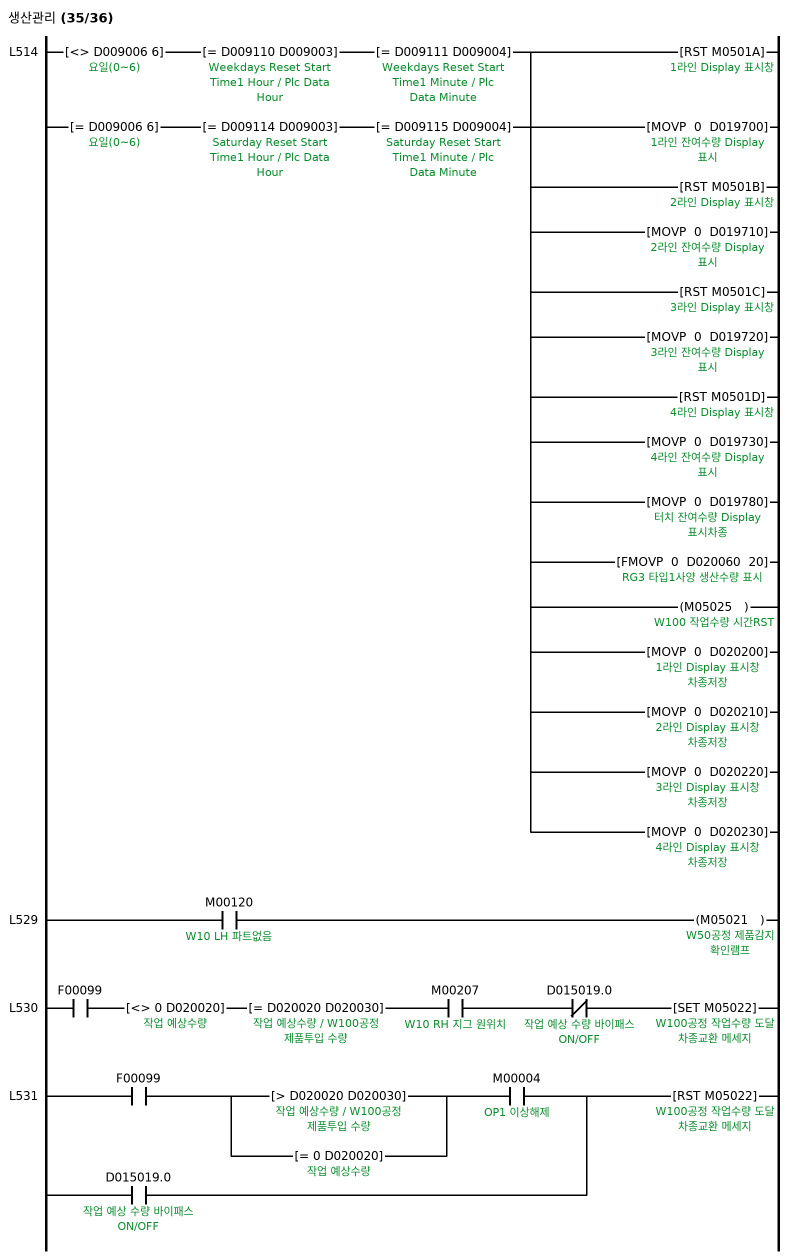
[picture p480: 생산관리 rungs L514-L531]
; L514
LOAD<>    D009006 6	// 요일(0~6)
AND=      D009110 D009003	// Weekdays Reset Start Time1 Hour / Plc Data Hour
AND=      D009111 D009004	// Weekdays Reset Start Time1 Minute / Plc Data Minute
LOAD=     D009006 6	// 요일(0~6)
AND=      D009114 D009003	// Saturday Reset Start Time1 Hour / Plc Data Hour
AND=      D009115 D009004	// Saturday Reset Start Time1 Minute / Plc Data Minute
OR LOAD
RST       M0501A	// 1라인 Display 표시창
MOVP      0 D019700	// 1라인 잔여수량 Display 표시 
RST       M0501B	// 2라인 Display 표시창
MOVP      0 D019710	// 2라인 잔여수량 Display 표시 
RST       M0501C	// 3라인 Display 표시창
MOVP      0 D019720	// 3라인 잔여수량 Display 표시 
RST       M0501D	// 4라인 Display 표시창
MOVP      0 D019730	// 4라인 잔여수량 Display 표시 
MOVP      0 D019780	// 터치 잔여수량 Display 표시차종
FMOVP     0 D020060 20	// RG3 타입1사양 생산수량 표시
OUT       M05025	// W100 작업수량 시간RST
MOVP      0 D020200	// 1라인 Display 표시창 차종저장
MOVP      0 D020210	// 2라인 Display 표시창 차종저장
MOVP      0 D020220	// 3라인 Display 표시창 차종저장
MOVP      0 D020230	// 4라인 Display 표시창 차종저장
; L529
LOAD      M00120	// W10 LH 파트없음
OUT       M05021	// W50공정 제품감지 확인램프
; L530
LOAD      F00099
AND<>     0 D020020	// 작업 예상수량
AND=      D020020 D020030	// 작업 예상수량 / W100공정 제품투입 수량
AND       M00207	// W10 RH 지그 원위치
AND NOT   D015019.0	// 작업 예상 수량 바이패스 ON/OFF
SET       M05022	// W100공정 작업수량 도달 차종교환 메세지
; L531
LOAD      F00099
LOAD>     D020020 D020030	// 작업 예상수량 / W100공정 제품투입 수량
OR=       0 D020020	// 작업 예상수량
AND LOAD
AND       M00004	// OP1 이상해제
OR        D015019.0	// 작업 예상 수량 바이패스 ON/OFF
RST       M05022	// W100공정 작업수량 도달 차종교환 메세지

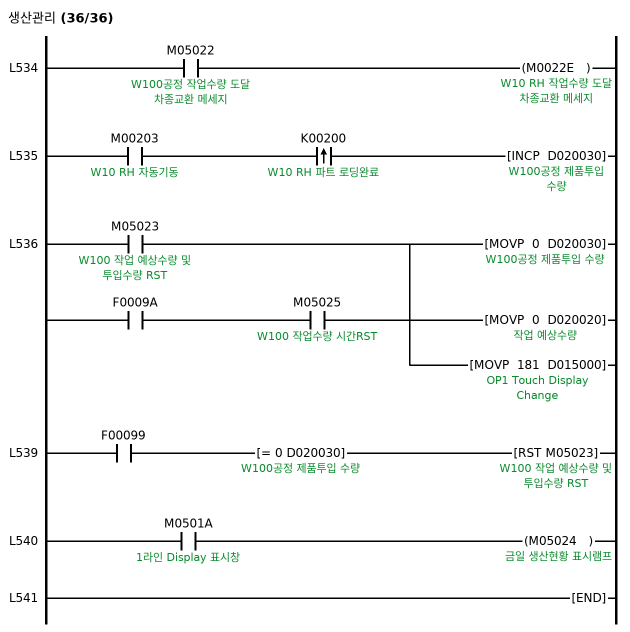
; L534
LOAD      M05022	// W100공정 작업수량 도달 차종교환 메세지
OUT       M0022E	// W10 RH 작업수량 도달 차종교환 메세지
; L535
LOAD      M00203	// W10 RH 자동기동
ANDP      K00200	// W10 RH 파트 로딩완료
INCP      D020030	// W100공정 제품투입 수량
; L536
LOAD      M05023	// W100 작업 예상수량 및 투입수량 RST
LOAD      F0009A
AND       M05025	// W100 작업수량 시간RST
OR LOAD
MOVP      0 D020030	// W100공정 제품투입 수량
MOVP      0 D020020	// 작업 예상수량
MOVP      181 D015000	// OP1 Touch Display Change
; L539
LOAD      F00099
AND=      0 D020030	// W100공정 제품투입 수량
RST       M05023	// W100 작업 예상수량 및 투입수량 RST
; L540
LOAD      M0501A	// 1라인 Display 표시창
OUT       M05024	// 금일 생산현황 표시램프
; L541
END

PROGRAM 생산현황판 (task: 스캔 프로그램)

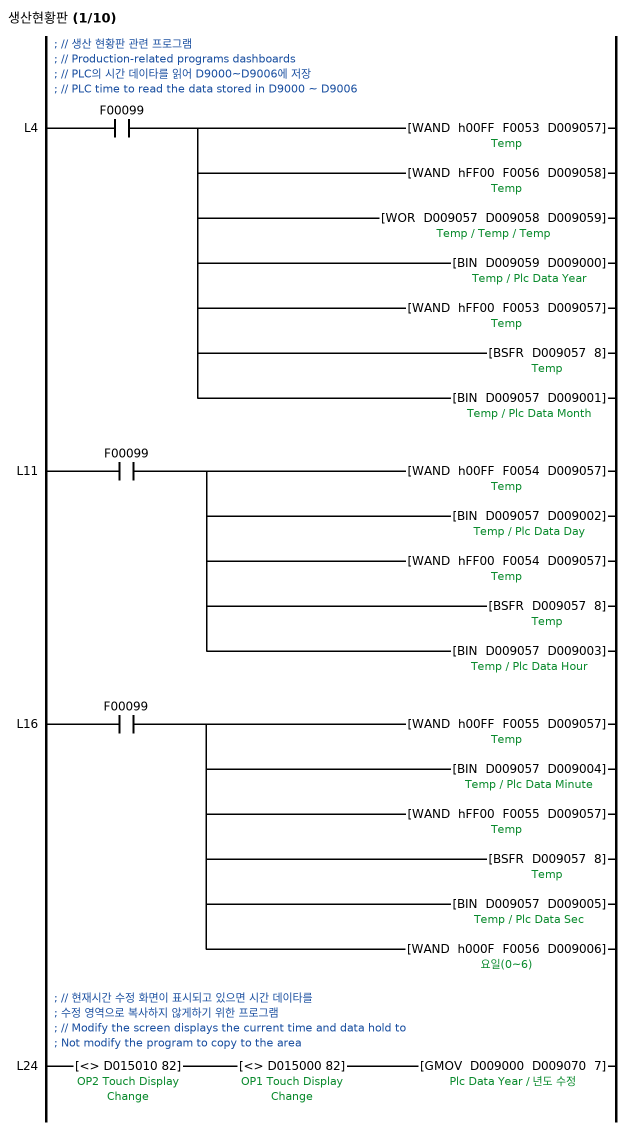
// // 생산 현황판 관련 프로그램
// // Production-related programs dashboards
//   // PLC의 시간 데이타를 읽어 D9000~D9006에 저장
//   // PLC time to read the data stored in D9000 ~ D9006
; L4
LOAD      F00099
WAND      h00FF F0053 D009057	// Temp
WAND      hFF00 F0056 D009058	// Temp
WOR       D009057 D009058 D009059	// Temp / Temp / Temp
BIN       D009059 D009000	// Temp / Plc Data Year
WAND      hFF00 F0053 D009057	// Temp
BSFR      D009057 8	// Temp
BIN       D009057 D009001	// Temp / Plc Data Month
; L11
LOAD      F00099
WAND      h00FF F0054 D009057	// Temp
BIN       D009057 D009002	// Temp / Plc Data Day
WAND      hFF00 F0054 D009057	// Temp
BSFR      D009057 8	// Temp
BIN       D009057 D009003	// Temp / Plc Data Hour
; L16
LOAD      F00099
WAND      h00FF F0055 D009057	// Temp
BIN       D009057 D009004	// Temp / Plc Data Minute
WAND      hFF00 F0055 D009057	// Temp
BSFR      D009057 8	// Temp
BIN       D009057 D009005	// Temp / Plc Data Sec
WAND      h000F F0056 D009006	// 요일(0~6)
//   // 현재시간 수정 화면이 표시되고 있으면 시간 데이타를
//      수정 영역으로 복사하지 않게하기 위한 프로그램
//   // Modify the screen displays the current time and data hold to
//       Not modify the program to copy to the area
; L24
LOAD<>    D015010 82	// OP2 Touch Display Change
AND<>     D015000 82	// OP1 Touch Display Change
GMOV      D009000 D009070 7	// Plc Data Year / 년도 수정

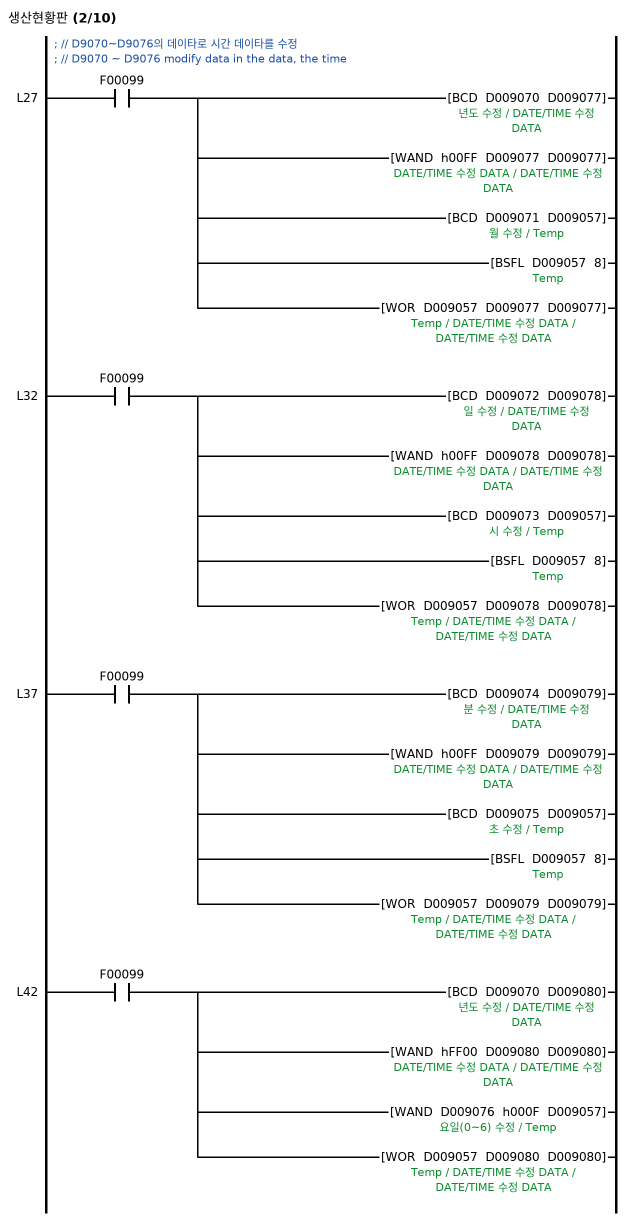
//   // D9070~D9076의 데이타로 시간 데이타를 수정
//   // D9070 ~ D9076 modify data in the data, the time
; L27
LOAD      F00099
BCD       D009070 D009077	// 년도 수정 / DATE/TIME 수정 DATA
WAND      h00FF D009077 D009077	// DATE/TIME 수정 DATA / DATE/TIME 수정 DATA
BCD       D009071 D009057	// 월 수정 / Temp
BSFL      D009057 8	// Temp
WOR       D009057 D009077 D009077	// Temp / DATE/TIME 수정 DATA / DATE/TIME 수정 DATA
; L32
LOAD      F00099
BCD       D009072 D009078	// 일 수정 / DATE/TIME 수정 DATA
WAND      h00FF D009078 D009078	// DATE/TIME 수정 DATA / DATE/TIME 수정 DATA
BCD       D009073 D009057	// 시 수정 / Temp
BSFL      D009057 8	// Temp
WOR       D009057 D009078 D009078	// Temp / DATE/TIME 수정 DATA / DATE/TIME 수정 DATA
; L37
LOAD      F00099
BCD       D009074 D009079	// 분 수정 / DATE/TIME 수정 DATA
WAND      h00FF D009079 D009079	// DATE/TIME 수정 DATA / DATE/TIME 수정 DATA
BCD       D009075 D009057	// 초 수정 / Temp
BSFL      D009057 8	// Temp
WOR       D009057 D009079 D009079	// Temp / DATE/TIME 수정 DATA / DATE/TIME 수정 DATA
; L42
LOAD      F00099
BCD       D009070 D009080	// 년도 수정 / DATE/TIME 수정 DATA
WAND      hFF00 D009080 D009080	// DATE/TIME 수정 DATA / DATE/TIME 수정 DATA
WAND      D009076 h000F D009057	// 요일(0~6) 수정 / Temp
WOR       D009057 D009080 D009080	// Temp / DATE/TIME 수정 DATA / DATE/TIME 수정 DATA

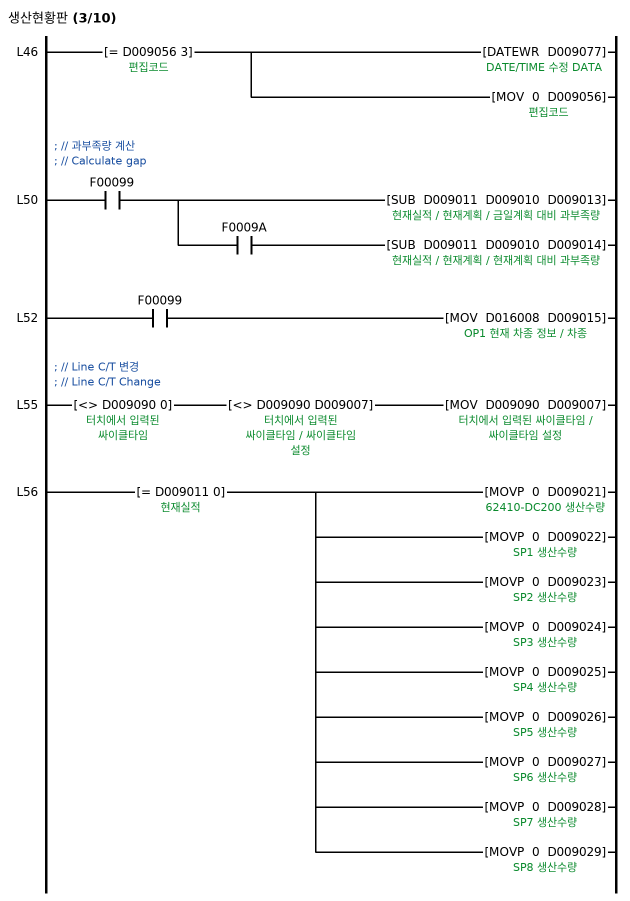
; L46
LOAD=     D009056 3	// 편집코드
DATEWR    D009077	// DATE/TIME 수정 DATA
MOV       0 D009056	// 편집코드
//   // 과부족량 계산
//   // Calculate gap
; L50
LOAD      F00099
SUB       D009011 D009010 D009013	// 현재실적 / 현재계획 / 금일계획 대비 과부족량
AND       F0009A
SUB       D009011 D009010 D009014	// 현재실적 / 현재계획 / 현재계획 대비 과부족량
; L52
LOAD      F00099
MOV       D016008 D009015	// OP1 현재 차종 정보 / 차종
//   // Line C/T 변경
//   // Line C/T Change
; L55
LOAD<>    D009090 0	// 터치에서 입력된 싸이클타임
AND<>     D009090 D009007	// 터치에서 입력된 싸이클타임 / 싸이클타임 설정
MOV       D009090 D009007	// 터치에서 입력된 싸이클타임 / 싸이클타임 설정
; L56
LOAD=     D009011 0	// 현재실적
MOVP      0 D009021	// 62410-DC200 생산수량
MOVP      0 D009022	// SP1 생산수량
MOVP      0 D009023	// SP2 생산수량
MOVP      0 D009024	// SP3 생산수량
MOVP      0 D009025	// SP4 생산수량
MOVP      0 D009026	// SP5 생산수량
MOVP      0 D009027	// SP6 생산수량
MOVP      0 D009028	// SP7 생산수량
MOVP      0 D009029	// SP8 생산수량

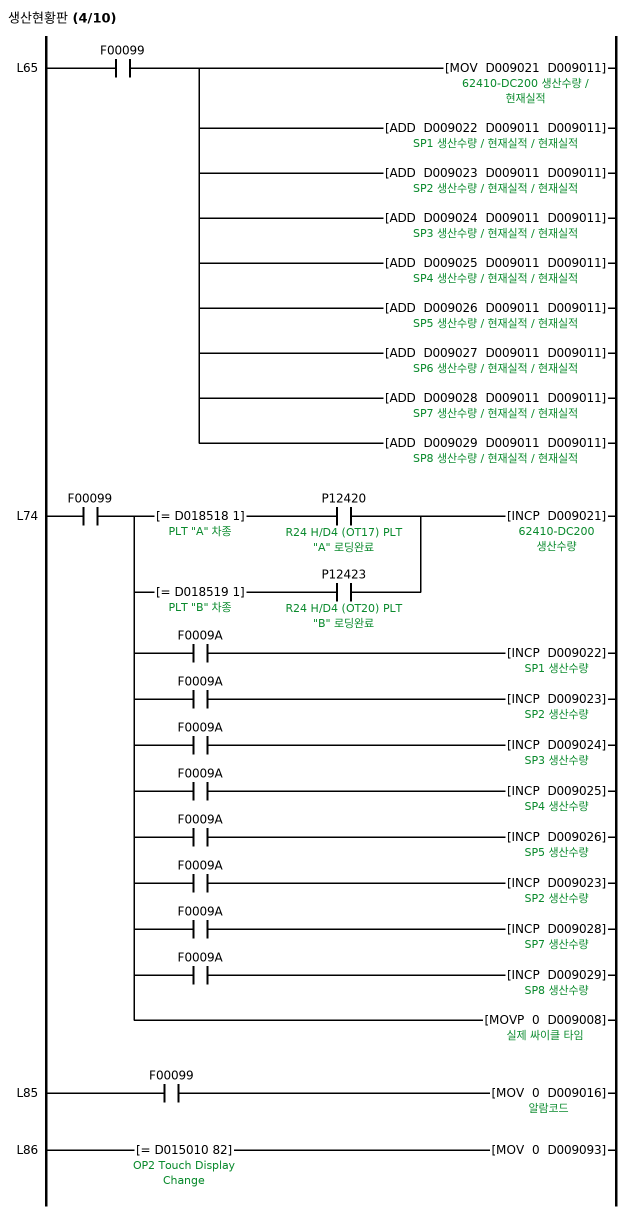
; L65
LOAD      F00099
MOV       D009021 D009011	// 62410-DC200 생산수량 / 현재실적
ADD       D009022 D009011 D009011	// SP1 생산수량 / 현재실적 / 현재실적
ADD       D009023 D009011 D009011	// SP2 생산수량 / 현재실적 / 현재실적
ADD       D009024 D009011 D009011	// SP3 생산수량 / 현재실적 / 현재실적
ADD       D009025 D009011 D009011	// SP4 생산수량 / 현재실적 / 현재실적
ADD       D009026 D009011 D009011	// SP5 생산수량 / 현재실적 / 현재실적
ADD       D009027 D009011 D009011	// SP6 생산수량 / 현재실적 / 현재실적
ADD       D009028 D009011 D009011	// SP7 생산수량 / 현재실적 / 현재실적
ADD       D009029 D009011 D009011	// SP8 생산수량 / 현재실적 / 현재실적
; L74
LOAD      F00099
MPUSH
LOAD=     D018518 1	// PLT "A" 차종
AND       P12420	// R24 H/D4 (OT17) PLT "A" 로딩완료
LOAD=     D018519 1	// PLT "B" 차종
AND       P12423	// R24 H/D4 (OT20) PLT "B" 로딩완료
OR LOAD
AND LOAD
INCP      D009021	// 62410-DC200 생산수량
MLOAD
AND       F0009A
INCP      D009022	// SP1 생산수량
MLOAD
AND       F0009A
INCP      D009023	// SP2 생산수량
MLOAD
AND       F0009A
INCP      D009024	// SP3 생산수량
MLOAD
AND       F0009A
INCP      D009025	// SP4 생산수량
MLOAD
AND       F0009A
INCP      D009026	// SP5 생산수량
MLOAD
AND       F0009A
INCP      D009023	// SP2 생산수량
MLOAD
AND       F0009A
INCP      D009028	// SP7 생산수량
MLOAD
AND       F0009A
INCP      D009029	// SP8 생산수량
MPOP
MOVP      0 D009008	// 실제 싸이클 타임
; L85
LOAD      F00099
MOV       0 D009016	// 알람코드
; L86
LOAD=     D015010 82	// OP2 Touch Display Change
MOV       0 D009093

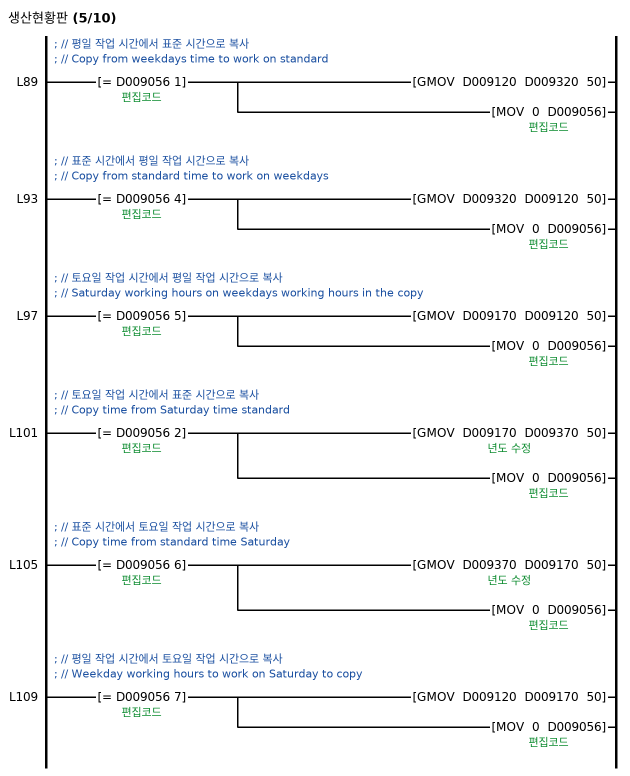
//   // 평일 작업 시간에서 표준 시간으로 복사
//   // Copy from weekdays time to work on standard
; L89
LOAD=     D009056 1	// 편집코드
GMOV      D009120 D009320 50
MOV       0 D009056	// 편집코드
//   // 표준 시간에서 평일 작업 시간으로 복사
//   // Copy from standard time to work on weekdays
; L93
LOAD=     D009056 4	// 편집코드
GMOV      D009320 D009120 50
MOV       0 D009056	// 편집코드
//   // 토요일 작업 시간에서 평일 작업 시간으로 복사
//   // Saturday working hours on weekdays working hours in the copy
; L97
LOAD=     D009056 5	// 편집코드
GMOV      D009170 D009120 50
MOV       0 D009056	// 편집코드
//   // 토요일 작업 시간에서 표준 시간으로 복사
//   // Copy time from Saturday time standard
; L101
LOAD=     D009056 2	// 편집코드
GMOV      D009170 D009370 50	// 년도 수정
MOV       0 D009056	// 편집코드
//   // 표준 시간에서 토요일 작업 시간으로 복사
//   // Copy time from standard time Saturday
; L105
LOAD=     D009056 6	// 편집코드
GMOV      D009370 D009170 50	// 년도 수정
MOV       0 D009056	// 편집코드
//   // 평일 작업 시간에서 토요일 작업 시간으로 복사
//   // Weekday working hours to work on Saturday to copy
; L109
LOAD=     D009056 7	// 편집코드
GMOV      D009120 D009170 50
MOV       0 D009056	// 편집코드

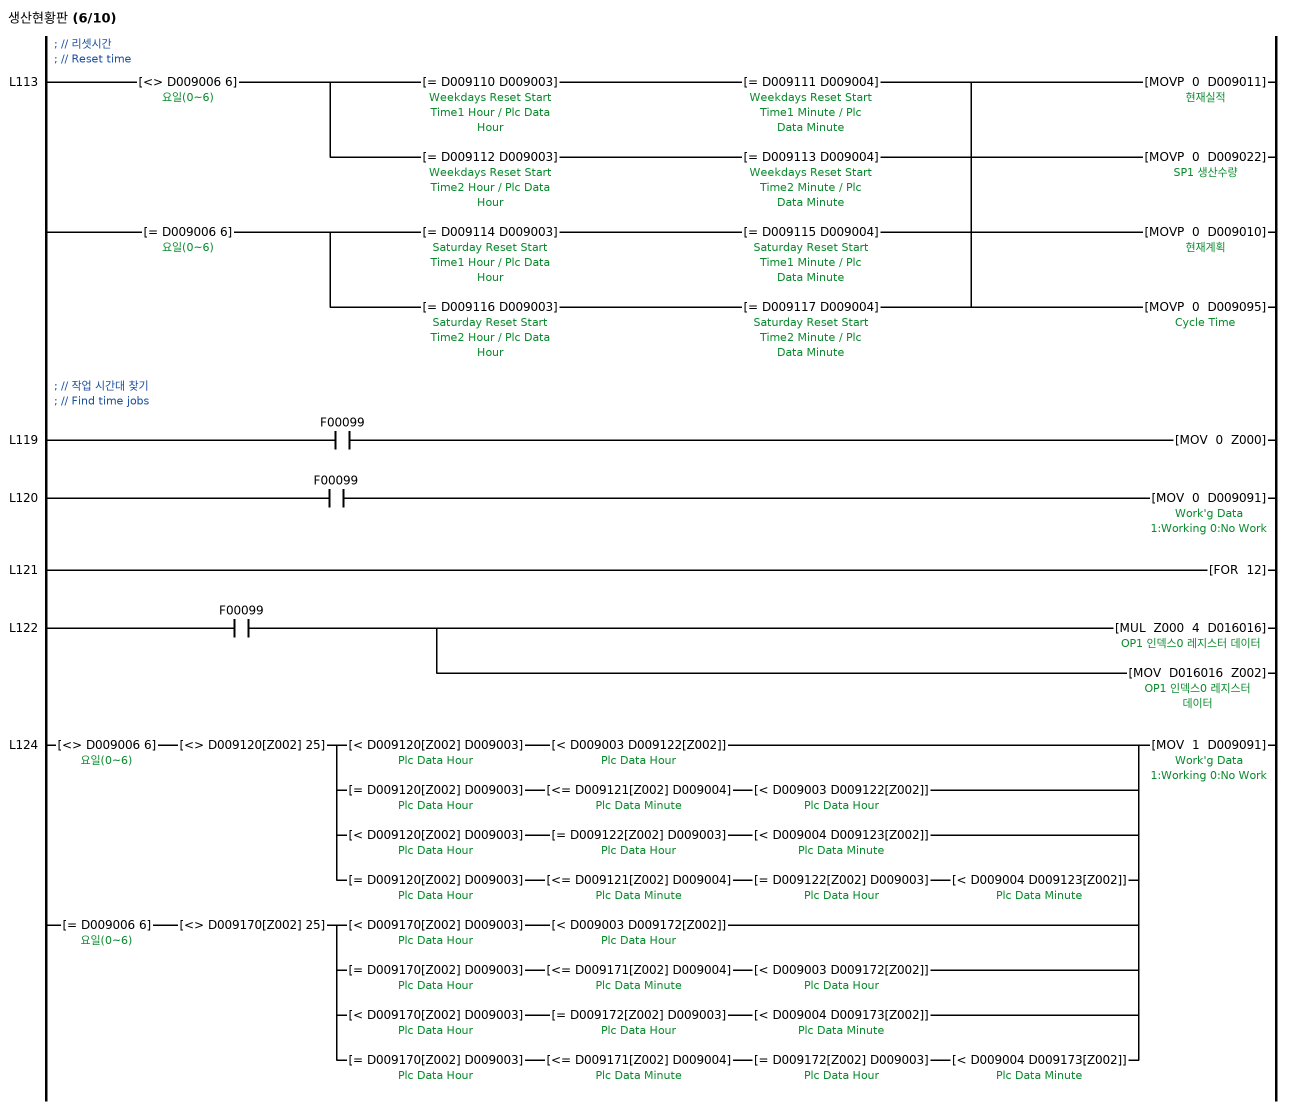
//   // 리셋시간
//   // Reset time
; L113
LOAD<>    D009006 6	// 요일(0~6)
LOAD=     D009110 D009003	// Weekdays Reset Start Time1 Hour / Plc Data Hour
AND=      D009111 D009004	// Weekdays Reset Start Time1 Minute / Plc Data Minute
LOAD=     D009112 D009003	// Weekdays Reset Start Time2 Hour / Plc Data Hour
AND=      D009113 D009004	// Weekdays Reset Start Time2 Minute / Plc Data Minute
OR LOAD
AND LOAD
LOAD=     D009006 6	// 요일(0~6)
LOAD=     D009114 D009003	// Saturday Reset Start Time1 Hour / Plc Data Hour
AND=      D009115 D009004	// Saturday Reset Start Time1 Minute / Plc Data Minute
LOAD=     D009116 D009003	// Saturday Reset Start Time2 Hour / Plc Data Hour
AND=      D009117 D009004	// Saturday Reset Start Time2 Minute / Plc Data Minute
OR LOAD
AND LOAD
OR LOAD
MOVP      0 D009011	// 현재실적
MOVP      0 D009022	// SP1 생산수량
MOVP      0 D009010	// 현재계획
MOVP      0 D009095	// Cycle Time
//   // 작업 시간대 찾기
//   // Find time jobs
; L119
LOAD      F00099
MOV       0 Z000
; L120
LOAD      F00099
MOV       0 D009091	// Work'g Data 1:Working 0:No Work
; L121
FOR       12
; L122
LOAD      F00099
MUL       Z000 4 D016016	// OP1 인덱스0 레지스터 데이터
MOV       D016016 Z002	// OP1 인덱스0 레지스터 데이터
; L124
LOAD<>    D009006 6	// 요일(0~6)
AND<>     D009120[Z002] 25
LOAD<     D009120[Z002] D009003	// Plc Data Hour
AND<      D009003 D009122[Z002]	// Plc Data Hour
LOAD=     D009120[Z002] D009003	// Plc Data Hour
AND<=     D009121[Z002] D009004	// Plc Data Minute
AND<      D009003 D009122[Z002]	// Plc Data Hour
OR LOAD
LOAD<     D009120[Z002] D009003	// Plc Data Hour
AND=      D009122[Z002] D009003	// Plc Data Hour
AND<      D009004 D009123[Z002]	// Plc Data Minute
OR LOAD
LOAD=     D009120[Z002] D009003	// Plc Data Hour
AND<=     D009121[Z002] D009004	// Plc Data Minute
AND=      D009122[Z002] D009003	// Plc Data Hour
AND<      D009004 D009123[Z002]	// Plc Data Minute
OR LOAD
AND LOAD
LOAD=     D009006 6	// 요일(0~6)
AND<>     D009170[Z002] 25
LOAD<     D009170[Z002] D009003	// Plc Data Hour
AND<      D009003 D009172[Z002]	// Plc Data Hour
LOAD=     D009170[Z002] D009003	// Plc Data Hour
AND<=     D009171[Z002] D009004	// Plc Data Minute
AND<      D009003 D009172[Z002]	// Plc Data Hour
OR LOAD
LOAD<     D009170[Z002] D009003	// Plc Data Hour
AND=      D009172[Z002] D009003	// Plc Data Hour
AND<      D009004 D009173[Z002]	// Plc Data Minute
OR LOAD
LOAD=     D009170[Z002] D009003	// Plc Data Hour
AND<=     D009171[Z002] D009004	// Plc Data Minute
AND=      D009172[Z002] D009003	// Plc Data Hour
AND<      D009004 D009173[Z002]	// Plc Data Minute
OR LOAD
AND LOAD
OR LOAD
MOV       1 D009091	// Work'g Data 1:Working 0:No Work

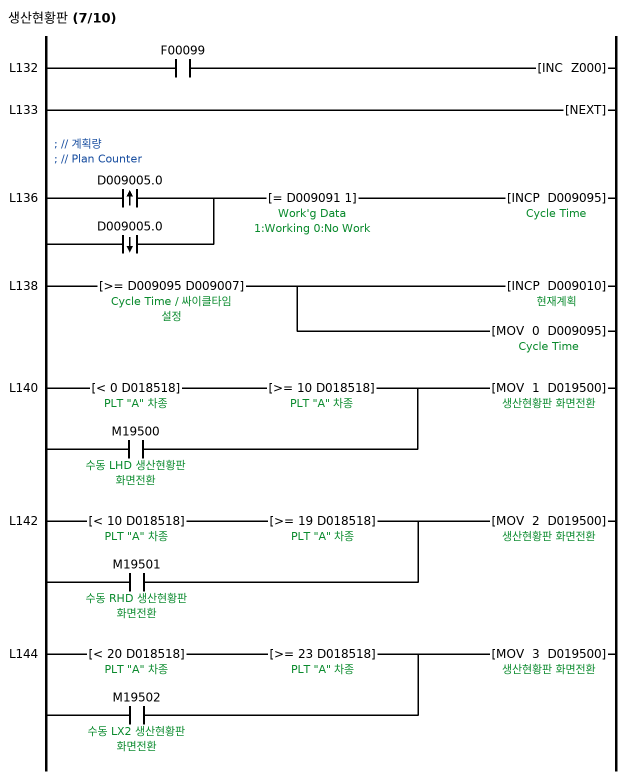
; L132
LOAD      F00099
INC       Z000
; L133
NEXT
// // 계획량
// // Plan Counter
; L136
LOADP     D009005.0
ORN       D009005.0
AND=      D009091 1	// Work'g Data 1:Working 0:No Work
INCP      D009095	// Cycle Time
; L138
LOAD>=    D009095 D009007	// Cycle Time / 싸이클타임 설정
INCP      D009010	// 현재계획
MOV       0 D009095	// Cycle Time
; L140
LOAD<     0 D018518	// PLT "A" 차종
AND>=     10 D018518	// PLT "A" 차종
OR        M19500	// 수동 LHD 생산현황판 화면전환
MOV       1 D019500	// 생산현황판 화면전환
; L142
LOAD<     10 D018518	// PLT "A" 차종
AND>=     19 D018518	// PLT "A" 차종
OR        M19501	// 수동 RHD 생산현황판 화면전환
MOV       2 D019500	// 생산현황판 화면전환
; L144
LOAD<     20 D018518	// PLT "A" 차종
AND>=     23 D018518	// PLT "A" 차종
OR        M19502	// 수동 LX2 생산현황판 화면전환
MOV       3 D019500	// 생산현황판 화면전환

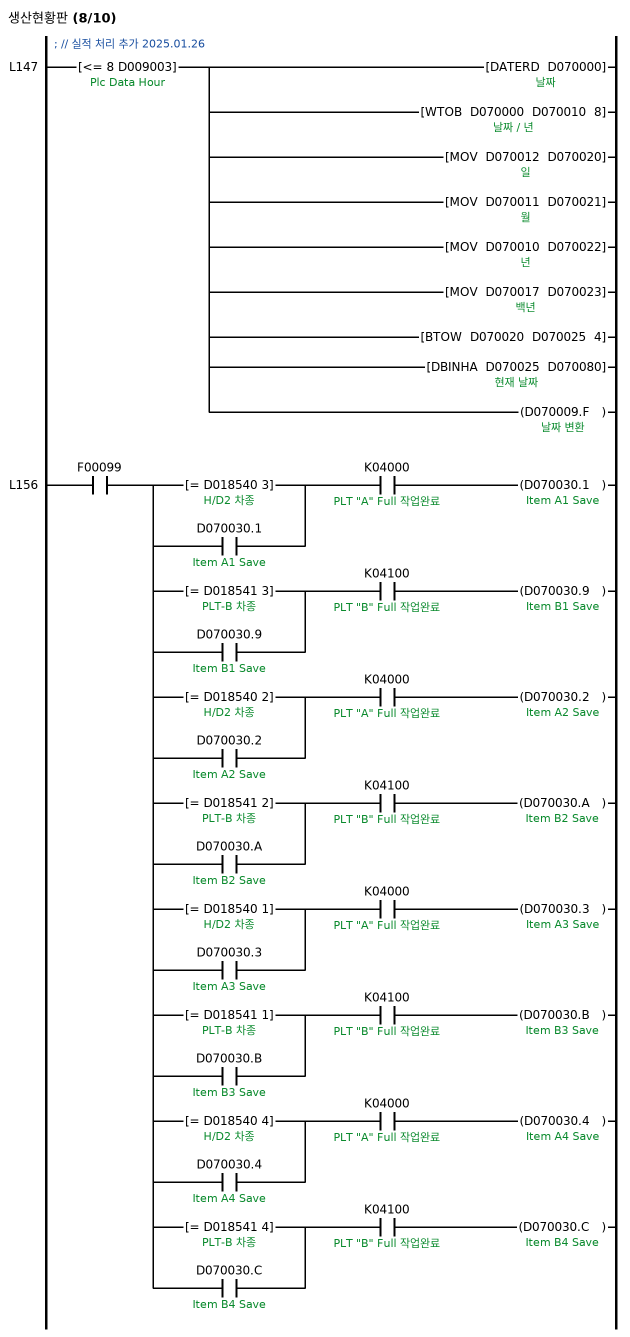
// // 실적 처리 추가 2025.01.26
; L147
LOAD<=    8 D009003	// Plc Data Hour
DATERD    D070000	// 날짜
WTOB      D070000 D070010 8	// 날짜 / 년
MOV       D070012 D070020	// 일
MOV       D070011 D070021	// 월
MOV       D070010 D070022	// 년
MOV       D070017 D070023	// 백년
BTOW      D070020 D070025 4
DBINHA    D070025 D070080	// 현재 날짜
OUT       D070009.F	// 날짜 변환
; L156
LOAD      F00099
MPUSH
LOAD=     D018540 3	// H/D2 차종
OR        D070030.1	// Item A1 Save
AND LOAD
AND       K04000	// PLT "A" Full 작업완료
OUT       D070030.1	// Item A1 Save
MLOAD
LOAD=     D018541 3	// PLT-B 차종
OR        D070030.9	// Item B1 Save
AND LOAD
AND       K04100	// PLT "B" Full 작업완료
OUT       D070030.9	// Item B1 Save
MLOAD
LOAD=     D018540 2	// H/D2 차종
OR        D070030.2	// Item A2 Save
AND LOAD
AND       K04000	// PLT "A" Full 작업완료
OUT       D070030.2	// Item A2 Save
MLOAD
LOAD=     D018541 2	// PLT-B 차종
OR        D070030.A	// Item B2 Save
AND LOAD
AND       K04100	// PLT "B" Full 작업완료
OUT       D070030.A	// Item B2 Save
MLOAD
LOAD=     D018540 1	// H/D2 차종
OR        D070030.3	// Item A3 Save
AND LOAD
AND       K04000	// PLT "A" Full 작업완료
OUT       D070030.3	// Item A3 Save
MLOAD
LOAD=     D018541 1	// PLT-B 차종
OR        D070030.B	// Item B3 Save
AND LOAD
AND       K04100	// PLT "B" Full 작업완료
OUT       D070030.B	// Item B3 Save
MLOAD
LOAD=     D018540 4	// H/D2 차종
OR        D070030.4	// Item A4 Save
AND LOAD
AND       K04000	// PLT "A" Full 작업완료
OUT       D070030.4	// Item A4 Save
MPOP
LOAD=     D018541 4	// PLT-B 차종
OR        D070030.C	// Item B4 Save
AND LOAD
AND       K04100	// PLT "B" Full 작업완료
OUT       D070030.C	// Item B4 Save

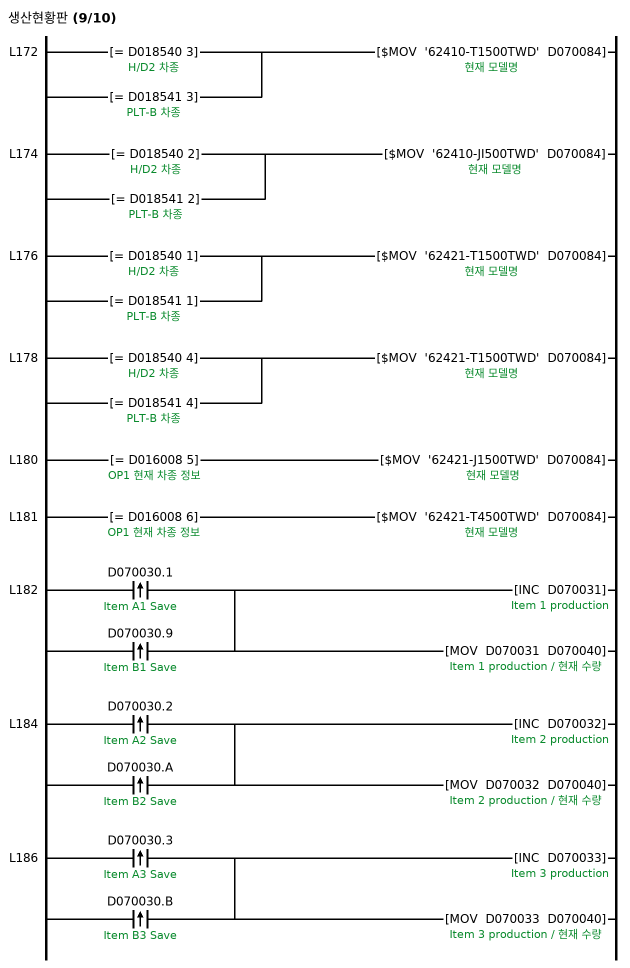
; L172
LOAD=     D018540 3	// H/D2 차종
OR=       D018541 3	// PLT-B 차종
$MOV      '62410-T1500TWD' D070084	// 현재 모델명
; L174
LOAD=     D018540 2	// H/D2 차종
OR=       D018541 2	// PLT-B 차종
$MOV      '62410-JI500TWD' D070084	// 현재 모델명
; L176
LOAD=     D018540 1	// H/D2 차종
OR=       D018541 1	// PLT-B 차종
$MOV      '62421-T1500TWD' D070084	// 현재 모델명
; L178
LOAD=     D018540 4	// H/D2 차종
OR=       D018541 4	// PLT-B 차종
$MOV      '62421-T1500TWD' D070084	// 현재 모델명
; L180
LOAD=     D016008 5	// OP1 현재 차종 정보
$MOV      '62421-J1500TWD' D070084	// 현재 모델명
; L181
LOAD=     D016008 6	// OP1 현재 차종 정보
$MOV      '62421-T4500TWD' D070084	// 현재 모델명
; L182
LOADP     D070030.1	// Item A1 Save
ORP       D070030.9	// Item B1 Save
INC       D070031	// Item 1 production
MOV       D070031 D070040	// Item 1 production / 현재 수량
; L184
LOADP     D070030.2	// Item A2 Save
ORP       D070030.A	// Item B2 Save
INC       D070032	// Item 2 production
MOV       D070032 D070040	// Item 2 production / 현재 수량
; L186
LOADP     D070030.3	// Item A3 Save
ORP       D070030.B	// Item B3 Save
INC       D070033	// Item 3 production
MOV       D070033 D070040	// Item 3 production / 현재 수량

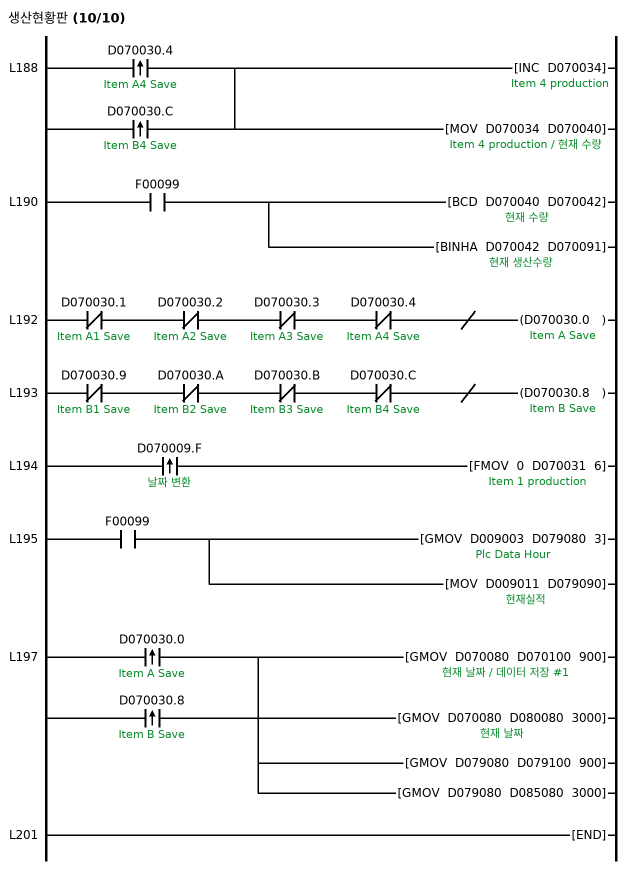
; L188
LOADP     D070030.4	// Item A4 Save
ORP       D070030.C	// Item B4 Save
INC       D070034	// Item 4 production
MOV       D070034 D070040	// Item 4 production / 현재 수량
; L190
LOAD      F00099
BCD       D070040 D070042	// 현재 수량
BINHA     D070042 D070091	// 현재 생산수량
; L192
LOAD NOT  D070030.1	// Item A1 Save
AND NOT   D070030.2	// Item A2 Save
AND NOT   D070030.3	// Item A3 Save
AND NOT   D070030.4	// Item A4 Save
NOT
OUT       D070030.0	// Item A Save
; L193
LOAD NOT  D070030.9	// Item B1 Save
AND NOT   D070030.A	// Item B2 Save
AND NOT   D070030.B	// Item B3 Save
AND NOT   D070030.C	// Item B4 Save
NOT
OUT       D070030.8	// Item B Save
; L194
LOADP     D070009.F	// 날짜 변환
FMOV      0 D070031 6	// Item 1 production
; L195
LOAD      F00099
GMOV      D009003 D079080 3	// Plc Data Hour
MOV       D009011 D079090	// 현재실적
; L197
LOADP     D070030.0	// Item A Save
ORP       D070030.8	// Item B Save
GMOV      D070080 D070100 900	// 현재 날짜 / 데이터 저장 #1
GMOV      D070080 D080080 3000	// 현재 날짜
GMOV      D079080 D079100 900
GMOV      D079080 D085080 3000
; L201
END

PROGRAM 판정데이터_트래킹 (task: 스캔 프로그램)

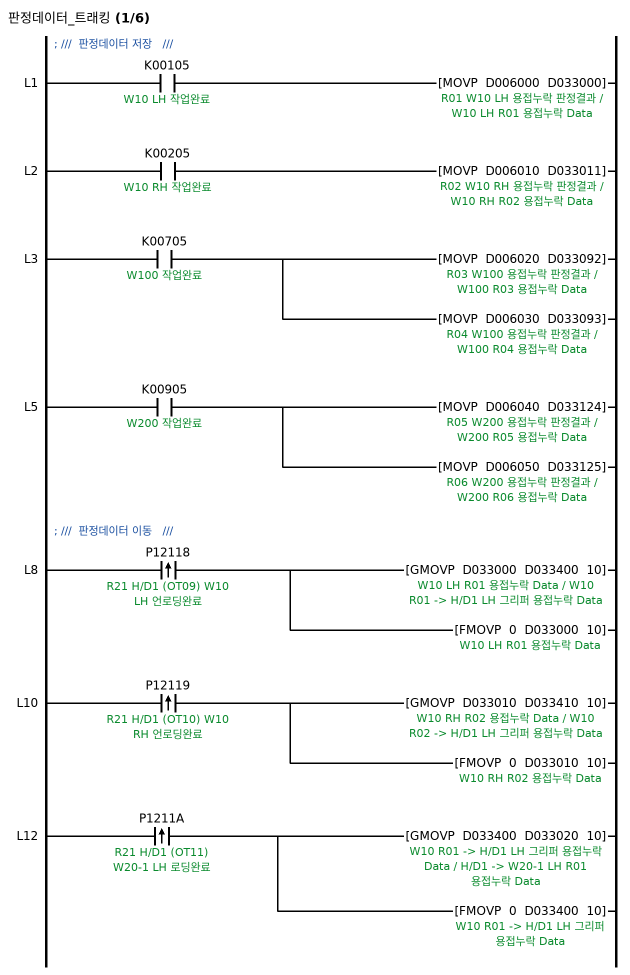
//    ///  판정데이터 저장   ///
; L1
LOAD      K00105	// W10 LH 작업완료
MOVP      D006000 D033000	// R01 W10 LH 용접누락 판정결과 / W10 LH R01 용접누락 Data
; L2
LOAD      K00205	// W10 RH 작업완료
MOVP      D006010 D033011	// R02 W10 RH 용접누락 판정결과 / W10 RH R02 용접누락 Data
; L3
LOAD      K00705	// W100 작업완료
MOVP      D006020 D033092	// R03 W100 용접누락 판정결과 / W100 R03 용접누락 Data
MOVP      D006030 D033093	// R04 W100 용접누락 판정결과 / W100 R04 용접누락 Data
; L5
LOAD      K00905	// W200 작업완료
MOVP      D006040 D033124	// R05 W200 용접누락 판정결과 / W200 R05 용접누락 Data
MOVP      D006050 D033125	// R06 W200 용접누락 판정결과 / W200 R06 용접누락 Data
//    ///  판정데이터 이동   ///
; L8
LOADP     P12118	// R21 H/D1 (OT09) W10 LH 언로딩완료
GMOVP     D033000 D033400 10	// W10 LH R01 용접누락 Data / W10 R01 -> H/D1 LH 그리퍼 용접누락 Data
FMOVP     0 D033000 10	// W10 LH R01 용접누락 Data
; L10
LOADP     P12119	// R21 H/D1 (OT10) W10 RH 언로딩완료
GMOVP     D033010 D033410 10	// W10 RH R02 용접누락 Data / W10 R02 -> H/D1 LH 그리퍼 용접누락 Data
FMOVP     0 D033010 10	// W10 RH R02 용접누락 Data
; L12
LOADP     P1211A	// R21 H/D1 (OT11) W20-1 LH 로딩완료
GMOVP     D033400 D033020 10	// W10 R01 -> H/D1 LH 그리퍼 용접누락 Data / H/D1 -> W20-1 LH R01 용접누락 Data
FMOVP     0 D033400 10	// W10 R01 -> H/D1 LH 그리퍼 용접누락 Data

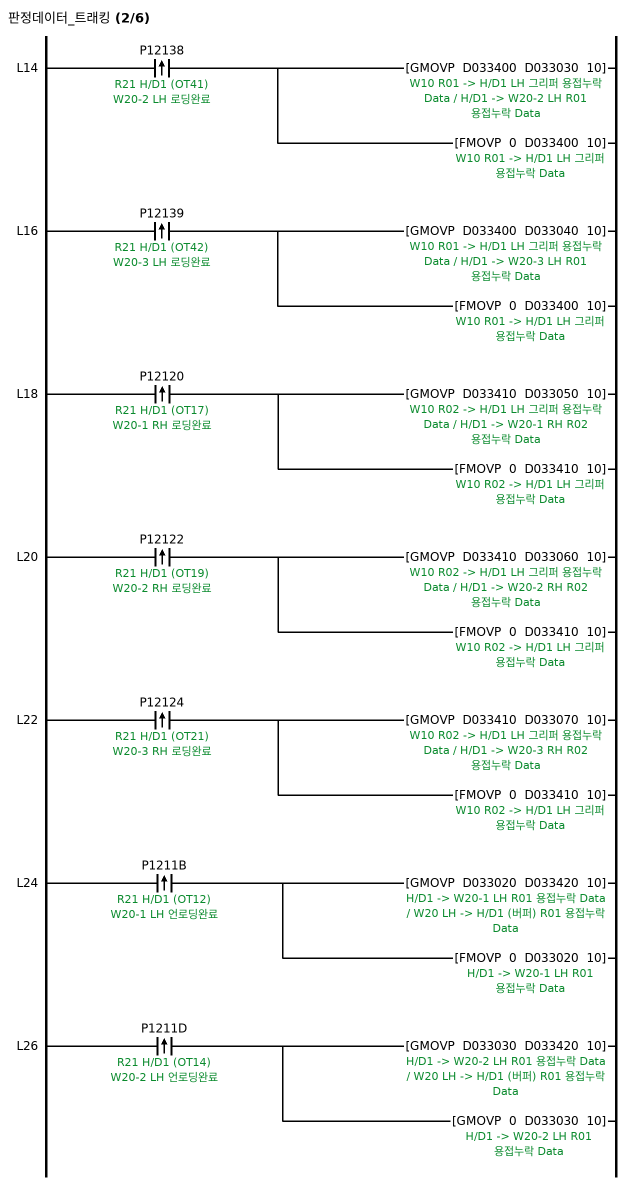
; L14
LOADP     P12138	// R21 H/D1 (OT41) W20-2 LH 로딩완료
GMOVP     D033400 D033030 10	// W10 R01 -> H/D1 LH 그리퍼 용접누락 Data / H/D1 -> W20-2 LH R01 용접누락 Data
FMOVP     0 D033400 10	// W10 R01 -> H/D1 LH 그리퍼 용접누락 Data
; L16
LOADP     P12139	// R21 H/D1 (OT42) W20-3 LH 로딩완료
GMOVP     D033400 D033040 10	// W10 R01 -> H/D1 LH 그리퍼 용접누락 Data / H/D1 -> W20-3 LH R01 용접누락 Data
FMOVP     0 D033400 10	// W10 R01 -> H/D1 LH 그리퍼 용접누락 Data
; L18
LOADP     P12120	// R21 H/D1 (OT17) W20-1 RH 로딩완료
GMOVP     D033410 D033050 10	// W10 R02 -> H/D1 LH 그리퍼 용접누락 Data / H/D1 -> W20-1 RH R02 용접누락 Data
FMOVP     0 D033410 10	// W10 R02 -> H/D1 LH 그리퍼 용접누락 Data
; L20
LOADP     P12122	// R21 H/D1 (OT19) W20-2 RH 로딩완료
GMOVP     D033410 D033060 10	// W10 R02 -> H/D1 LH 그리퍼 용접누락 Data / H/D1 -> W20-2 RH R02 용접누락 Data
FMOVP     0 D033410 10	// W10 R02 -> H/D1 LH 그리퍼 용접누락 Data
; L22
LOADP     P12124	// R21 H/D1 (OT21) W20-3 RH 로딩완료
GMOVP     D033410 D033070 10	// W10 R02 -> H/D1 LH 그리퍼 용접누락 Data / H/D1 -> W20-3 RH R02 용접누락 Data
FMOVP     0 D033410 10	// W10 R02 -> H/D1 LH 그리퍼 용접누락 Data
; L24
LOADP     P1211B	// R21 H/D1 (OT12) W20-1 LH 언로딩완료
GMOVP     D033020 D033420 10	// H/D1 -> W20-1 LH R01 용접누락 Data / W20 LH -> H/D1 (버퍼) R01 용접누락 Data
FMOVP     0 D033020 10	// H/D1 -> W20-1 LH R01 용접누락 Data
; L26
LOADP     P1211D	// R21 H/D1 (OT14) W20-2 LH 언로딩완료
GMOVP     D033030 D033420 10	// H/D1 -> W20-2 LH R01 용접누락 Data / W20 LH -> H/D1 (버퍼) R01 용접누락 Data
GMOVP     0 D033030 10	// H/D1 -> W20-2 LH R01 용접누락 Data

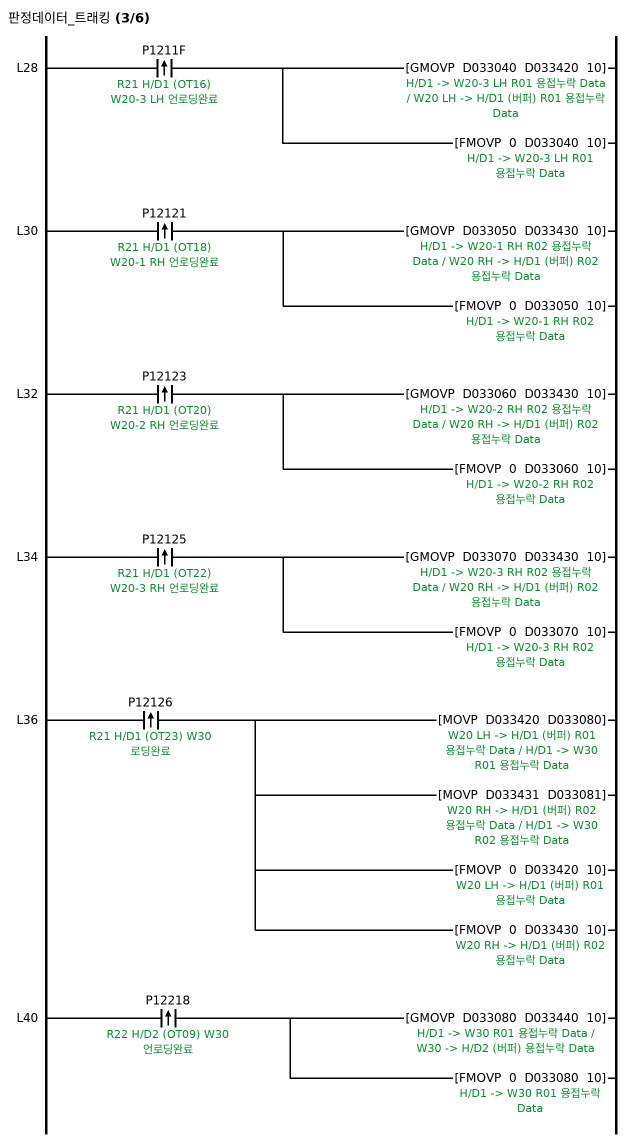
; L28
LOADP     P1211F	// R21 H/D1 (OT16) W20-3 LH 언로딩완료
GMOVP     D033040 D033420 10	// H/D1 -> W20-3 LH R01 용접누락 Data / W20 LH -> H/D1 (버퍼) R01 용접누락 Data
FMOVP     0 D033040 10	// H/D1 -> W20-3 LH R01 용접누락 Data
; L30
LOADP     P12121	// R21 H/D1 (OT18) W20-1 RH 언로딩완료
GMOVP     D033050 D033430 10	// H/D1 -> W20-1 RH R02 용접누락 Data / W20 RH -> H/D1 (버퍼) R02 용접누락 Data
FMOVP     0 D033050 10	// H/D1 -> W20-1 RH R02 용접누락 Data
; L32
LOADP     P12123	// R21 H/D1 (OT20) W20-2 RH 언로딩완료
GMOVP     D033060 D033430 10	// H/D1 -> W20-2 RH R02 용접누락 Data / W20 RH -> H/D1 (버퍼) R02 용접누락 Data
FMOVP     0 D033060 10	// H/D1 -> W20-2 RH R02 용접누락 Data
; L34
LOADP     P12125	// R21 H/D1 (OT22) W20-3 RH 언로딩완료
GMOVP     D033070 D033430 10	// H/D1 -> W20-3 RH R02 용접누락 Data / W20 RH -> H/D1 (버퍼) R02 용접누락 Data
FMOVP     0 D033070 10	// H/D1 -> W20-3 RH R02 용접누락 Data
; L36
LOADP     P12126	// R21 H/D1 (OT23) W30 로딩완료
MOVP      D033420 D033080	// W20 LH -> H/D1 (버퍼) R01 용접누락 Data / H/D1 -> W30 R01 용접누락 Data
MOVP      D033431 D033081	// W20 RH -> H/D1 (버퍼) R02 용접누락 Data / H/D1 -> W30 R02 용접누락 Data
FMOVP     0 D033420 10	// W20 LH -> H/D1 (버퍼) R01 용접누락 Data
FMOVP     0 D033430 10	// W20 RH -> H/D1 (버퍼) R02 용접누락 Data
; L40
LOADP     P12218	// R22 H/D2 (OT09) W30 언로딩완료
GMOVP     D033080 D033440 10	// H/D1 -> W30 R01 용접누락 Data / W30 -> H/D2 (버퍼) 용접누락 Data
FMOVP     0 D033080 10	// H/D1 -> W30 R01 용접누락 Data

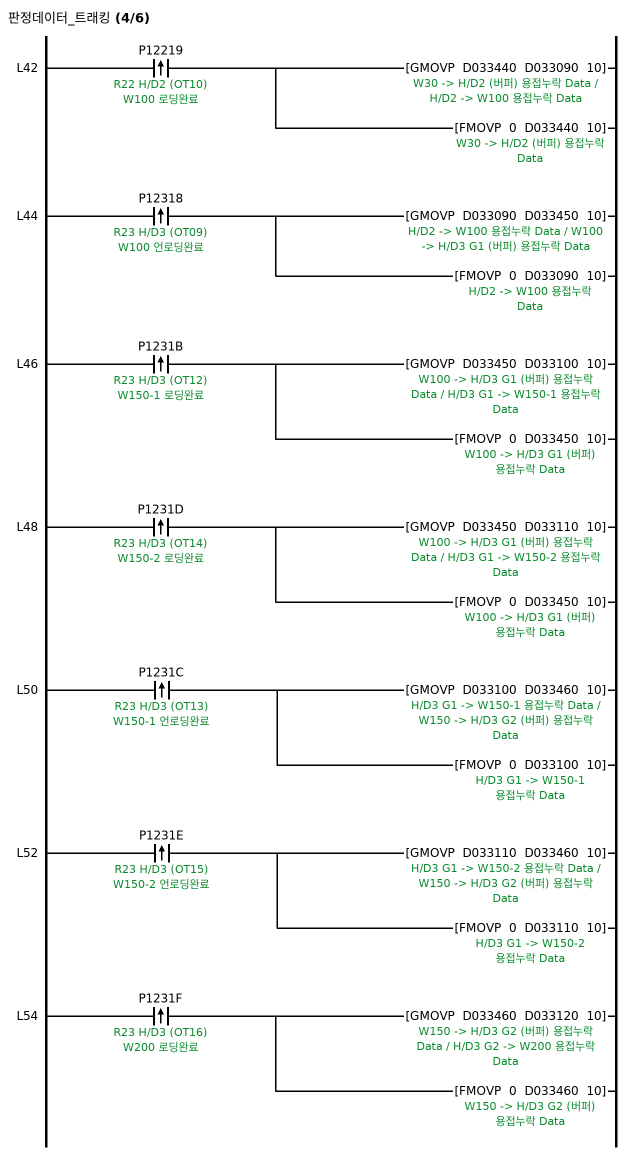
; L42
LOADP     P12219	// R22 H/D2 (OT10) W100 로딩완료
GMOVP     D033440 D033090 10	// W30 -> H/D2 (버퍼) 용접누락 Data / H/D2 -> W100 용접누락 Data
FMOVP     0 D033440 10	// W30 -> H/D2 (버퍼) 용접누락 Data
; L44
LOADP     P12318	// R23 H/D3 (OT09) W100 언로딩완료
GMOVP     D033090 D033450 10	// H/D2 -> W100 용접누락 Data / W100 -> H/D3 G1 (버퍼) 용접누락 Data
FMOVP     0 D033090 10	// H/D2 -> W100 용접누락 Data
; L46
LOADP     P1231B	// R23 H/D3 (OT12) W150-1 로딩완료
GMOVP     D033450 D033100 10	// W100 -> H/D3 G1 (버퍼) 용접누락 Data / H/D3 G1 -> W150-1 용접누락 Data
FMOVP     0 D033450 10	// W100 -> H/D3 G1 (버퍼) 용접누락 Data
; L48
LOADP     P1231D	// R23 H/D3 (OT14) W150-2 로딩완료
GMOVP     D033450 D033110 10	// W100 -> H/D3 G1 (버퍼) 용접누락 Data / H/D3 G1 -> W150-2 용접누락 Data
FMOVP     0 D033450 10	// W100 -> H/D3 G1 (버퍼) 용접누락 Data
; L50
LOADP     P1231C	// R23 H/D3 (OT13) W150-1 언로딩완료
GMOVP     D033100 D033460 10	// H/D3 G1 -> W150-1 용접누락 Data / W150 -> H/D3 G2 (버퍼) 용접누락 Data
FMOVP     0 D033100 10	// H/D3 G1 -> W150-1 용접누락 Data
; L52
LOADP     P1231E	// R23 H/D3 (OT15) W150-2 언로딩완료
GMOVP     D033110 D033460 10	// H/D3 G1 -> W150-2 용접누락 Data / W150 -> H/D3 G2 (버퍼) 용접누락 Data
FMOVP     0 D033110 10	// H/D3 G1 -> W150-2 용접누락 Data
; L54
LOADP     P1231F	// R23 H/D3 (OT16) W200 로딩완료
GMOVP     D033460 D033120 10	// W150 -> H/D3 G2 (버퍼) 용접누락 Data / H/D3 G2 -> W200 용접누락 Data
FMOVP     0 D033460 10	// W150 -> H/D3 G2 (버퍼) 용접누락 Data

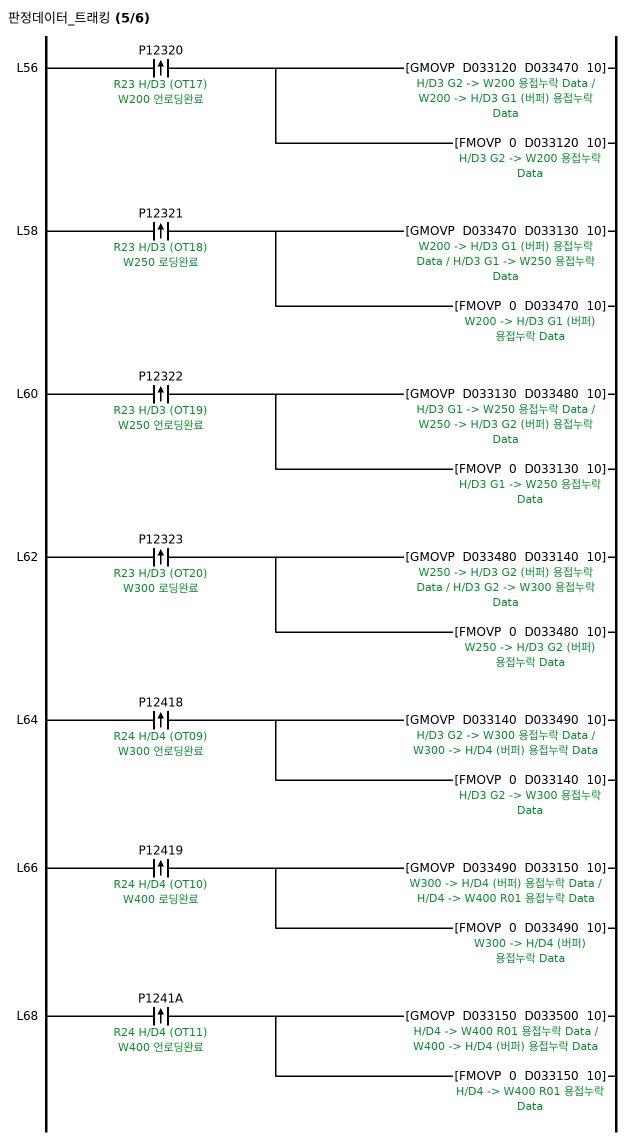
; L56
LOADP     P12320	// R23 H/D3 (OT17) W200 언로딩완료
GMOVP     D033120 D033470 10	// H/D3 G2 -> W200 용접누락 Data / W200 -> H/D3 G1 (버퍼) 용접누락 Data
FMOVP     0 D033120 10	// H/D3 G2 -> W200 용접누락 Data
; L58
LOADP     P12321	// R23 H/D3 (OT18) W250 로딩완료
GMOVP     D033470 D033130 10	// W200 -> H/D3 G1 (버퍼) 용접누락 Data / H/D3 G1 -> W250 용접누락 Data
FMOVP     0 D033470 10	// W200 -> H/D3 G1 (버퍼) 용접누락 Data
; L60
LOADP     P12322	// R23 H/D3 (OT19) W250 언로딩완료
GMOVP     D033130 D033480 10	// H/D3 G1 -> W250 용접누락 Data / W250 -> H/D3 G2 (버퍼) 용접누락 Data
FMOVP     0 D033130 10	// H/D3 G1 -> W250 용접누락 Data
; L62
LOADP     P12323	// R23 H/D3 (OT20) W300 로딩완료
GMOVP     D033480 D033140 10	// W250 -> H/D3 G2 (버퍼) 용접누락 Data / H/D3 G2 -> W300 용접누락 Data
FMOVP     0 D033480 10	// W250 -> H/D3 G2 (버퍼) 용접누락 Data
; L64
LOADP     P12418	// R24 H/D4 (OT09) W300 언로딩완료
GMOVP     D033140 D033490 10	// H/D3 G2 -> W300 용접누락 Data / W300 -> H/D4 (버퍼) 용접누락 Data
FMOVP     0 D033140 10	// H/D3 G2 -> W300 용접누락 Data
; L66
LOADP     P12419	// R24 H/D4 (OT10) W400 로딩완료
GMOVP     D033490 D033150 10	// W300 -> H/D4 (버퍼) 용접누락 Data / H/D4 -> W400 R01 용접누락 Data
FMOVP     0 D033490 10	// W300 -> H/D4 (버퍼) 용접누락 Data
; L68
LOADP     P1241A	// R24 H/D4 (OT11) W400 언로딩완료
GMOVP     D033150 D033500 10	// H/D4 -> W400 R01 용접누락 Data / W400 -> H/D4 (버퍼) 용접누락 Data
FMOVP     0 D033150 10	// H/D4 -> W400 R01 용접누락 Data

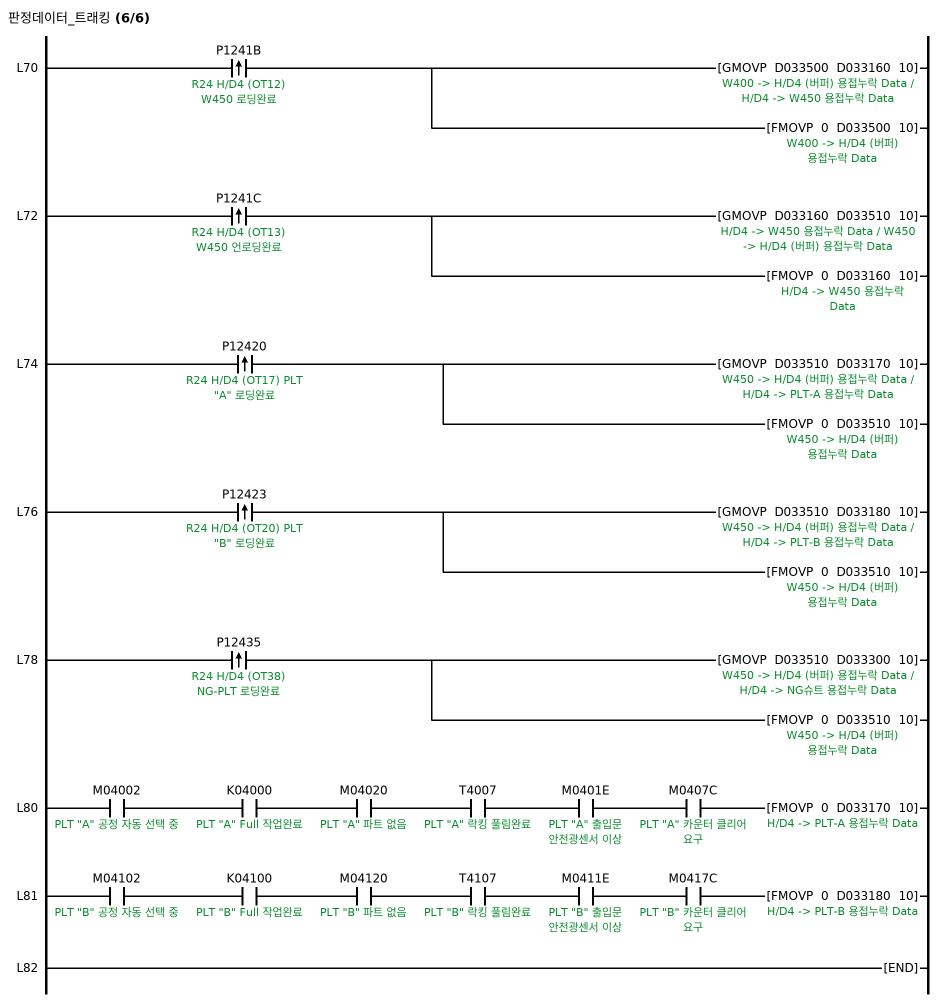
; L70
LOADP     P1241B	// R24 H/D4 (OT12) W450 로딩완료
GMOVP     D033500 D033160 10	// W400 -> H/D4 (버퍼) 용접누락 Data / H/D4 -> W450 용접누락 Data
FMOVP     0 D033500 10	// W400 -> H/D4 (버퍼) 용접누락 Data
; L72
LOADP     P1241C	// R24 H/D4 (OT13) W450 언로딩완료
GMOVP     D033160 D033510 10	// H/D4 -> W450 용접누락 Data / W450 -> H/D4 (버퍼) 용접누락 Data
FMOVP     0 D033160 10	// H/D4 -> W450 용접누락 Data
; L74
LOADP     P12420	// R24 H/D4 (OT17) PLT "A" 로딩완료
GMOVP     D033510 D033170 10	// W450 -> H/D4 (버퍼) 용접누락 Data / H/D4 -> PLT-A 용접누락 Data
FMOVP     0 D033510 10	// W450 -> H/D4 (버퍼) 용접누락 Data
; L76
LOADP     P12423	// R24 H/D4 (OT20) PLT "B" 로딩완료
GMOVP     D033510 D033180 10	// W450 -> H/D4 (버퍼) 용접누락 Data / H/D4 -> PLT-B 용접누락 Data
FMOVP     0 D033510 10	// W450 -> H/D4 (버퍼) 용접누락 Data
; L78
LOADP     P12435	// R24 H/D4 (OT38) NG-PLT 로딩완료
GMOVP     D033510 D033300 10	// W450 -> H/D4 (버퍼) 용접누락 Data / H/D4 -> NG슈트 용접누락 Data
FMOVP     0 D033510 10	// W450 -> H/D4 (버퍼) 용접누락 Data
; L80
LOAD      M04002	// PLT "A" 공정 자동 선택 중
AND       K04000	// PLT "A" Full 작업완료
AND       M04020	// PLT "A" 파트 없음
AND       T4007	// PLT "A" 락킹 풀림완료
AND       M0401E	// PLT "A" 출입문 안전광센서 이상
AND       M0407C	// PLT "A" 카운터 클리어 요구
FMOVP     0 D033170 10	// H/D4 -> PLT-A 용접누락 Data
; L81
LOAD      M04102	// PLT "B" 공정 자동 선택 중
AND       K04100	// PLT "B" Full 작업완료
AND       M04120	// PLT "B" 파트 없음
AND       T4107	// PLT "B" 락킹 풀림완료
AND       M0411E	// PLT "B" 출입문 안전광센서 이상
AND       M0417C	// PLT "B" 카운터 클리어 요구
FMOVP     0 D033180 10	// H/D4 -> PLT-B 용접누락 Data
; L82
END

PROGRAM 가스메타 (task: 스캔 프로그램)

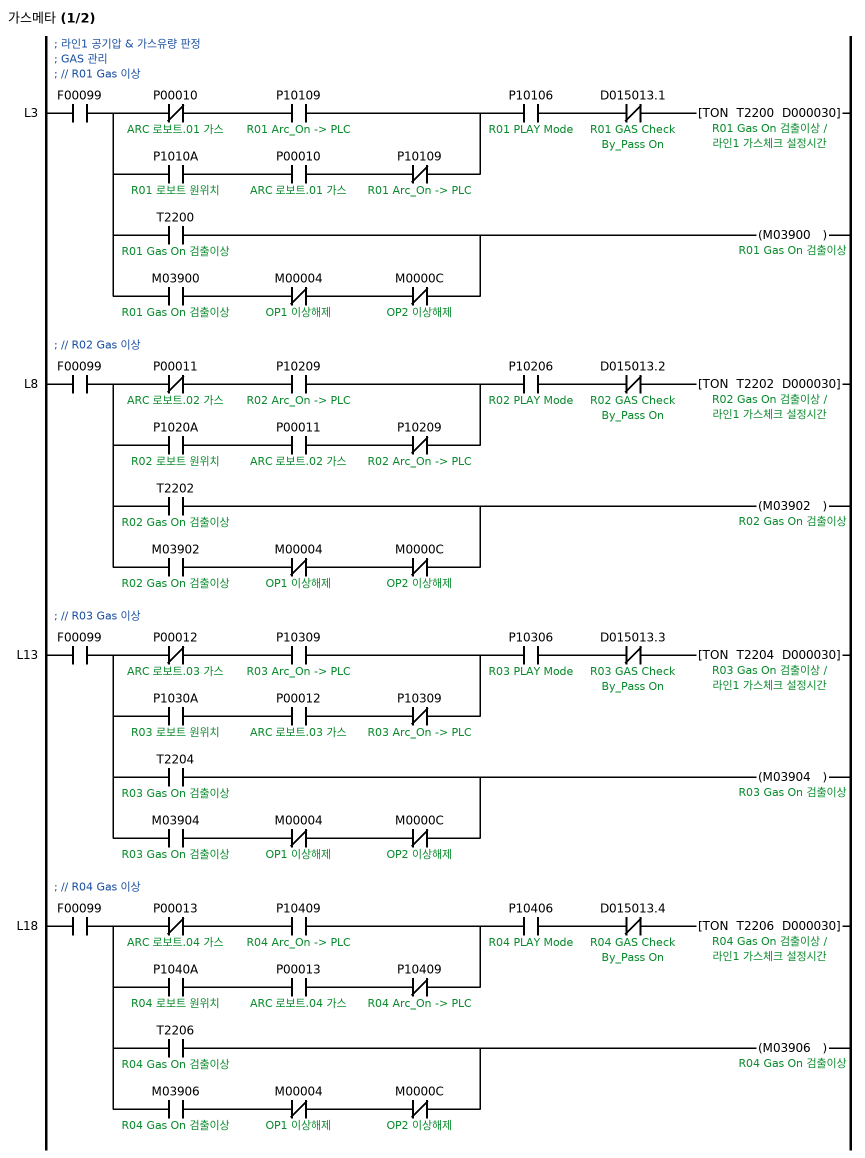
// 라인1 공기압 & 가스유량 판정
// GAS 관리
// // R01 Gas 이상
; L3
LOAD      F00099
MPUSH
LOAD NOT  P00010	// ARC 로보트.01 가스
AND       P10109	// R01 Arc_On -> PLC
LOAD      P1010A	// R01 로보트 원위치
AND       P00010	// ARC 로보트.01 가스
AND NOT   P10109	// R01 Arc_On -> PLC
OR LOAD
AND LOAD
AND       P10106	// R01 PLAY Mode
AND NOT   D015013.1	// R01 GAS Check By_Pass On
TON       T2200 D000030	// R01 Gas On 검출이상 / 라인1 가스체크 설정시간
MPOP
LOAD      T2200	// R01 Gas On 검출이상
LOAD      M03900	// R01 Gas On 검출이상
AND NOT   M00004	// OP1 이상해제
AND NOT   M0000C	// OP2 이상해제
OR LOAD
AND LOAD
OUT       M03900	// R01 Gas On 검출이상
// // R02 Gas 이상
; L8
LOAD      F00099
MPUSH
LOAD NOT  P00011	// ARC 로보트.02 가스
AND       P10209	// R02 Arc_On -> PLC
LOAD      P1020A	// R02 로보트 원위치
AND       P00011	// ARC 로보트.02 가스
AND NOT   P10209	// R02 Arc_On -> PLC
OR LOAD
AND LOAD
AND       P10206	// R02 PLAY Mode
AND NOT   D015013.2	// R02 GAS Check By_Pass On
TON       T2202 D000030	// R02 Gas On 검출이상 / 라인1 가스체크 설정시간
MPOP
LOAD      T2202	// R02 Gas On 검출이상
LOAD      M03902	// R02 Gas On 검출이상
AND NOT   M00004	// OP1 이상해제
AND NOT   M0000C	// OP2 이상해제
OR LOAD
AND LOAD
OUT       M03902	// R02 Gas On 검출이상
// // R03 Gas 이상
; L13
LOAD      F00099
MPUSH
LOAD NOT  P00012	// ARC 로보트.03 가스
AND       P10309	// R03 Arc_On -> PLC
LOAD      P1030A	// R03 로보트 원위치
AND       P00012	// ARC 로보트.03 가스
AND NOT   P10309	// R03 Arc_On -> PLC
OR LOAD
AND LOAD
AND       P10306	// R03 PLAY Mode
AND NOT   D015013.3	// R03 GAS Check By_Pass On
TON       T2204 D000030	// R03 Gas On 검출이상 / 라인1 가스체크 설정시간
MPOP
LOAD      T2204	// R03 Gas On 검출이상
LOAD      M03904	// R03 Gas On 검출이상
AND NOT   M00004	// OP1 이상해제
AND NOT   M0000C	// OP2 이상해제
OR LOAD
AND LOAD
OUT       M03904	// R03 Gas On 검출이상
// // R04 Gas 이상
; L18
LOAD      F00099
MPUSH
LOAD NOT  P00013	// ARC 로보트.04 가스
AND       P10409	// R04 Arc_On -> PLC
LOAD      P1040A	// R04 로보트 원위치
AND       P00013	// ARC 로보트.04 가스
AND NOT   P10409	// R04 Arc_On -> PLC
OR LOAD
AND LOAD
AND       P10406	// R04 PLAY Mode
AND NOT   D015013.4	// R04 GAS Check By_Pass On
TON       T2206 D000030	// R04 Gas On 검출이상 / 라인1 가스체크 설정시간
MPOP
LOAD      T2206	// R04 Gas On 검출이상
LOAD      M03906	// R04 Gas On 검출이상
AND NOT   M00004	// OP1 이상해제
AND NOT   M0000C	// OP2 이상해제
OR LOAD
AND LOAD
OUT       M03906	// R04 Gas On 검출이상

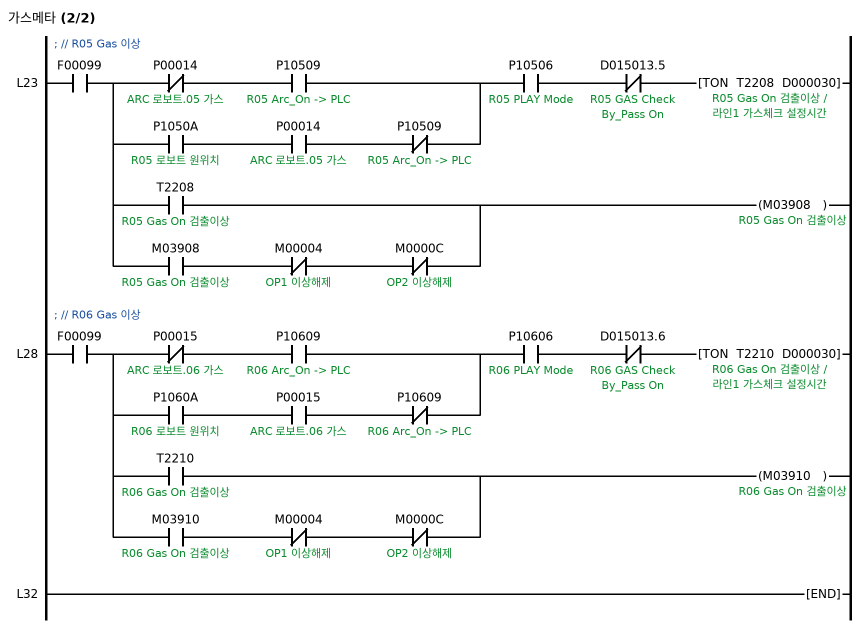
// // R05 Gas 이상
; L23
LOAD      F00099
MPUSH
LOAD NOT  P00014	// ARC 로보트.05 가스
AND       P10509	// R05 Arc_On -> PLC
LOAD      P1050A	// R05 로보트 원위치
AND       P00014	// ARC 로보트.05 가스
AND NOT   P10509	// R05 Arc_On -> PLC
OR LOAD
AND LOAD
AND       P10506	// R05 PLAY Mode
AND NOT   D015013.5	// R05 GAS Check By_Pass On
TON       T2208 D000030	// R05 Gas On 검출이상 / 라인1 가스체크 설정시간
MPOP
LOAD      T2208	// R05 Gas On 검출이상
LOAD      M03908	// R05 Gas On 검출이상
AND NOT   M00004	// OP1 이상해제
AND NOT   M0000C	// OP2 이상해제
OR LOAD
AND LOAD
OUT       M03908	// R05 Gas On 검출이상
// // R06 Gas 이상
; L28
LOAD      F00099
MPUSH
LOAD NOT  P00015	// ARC 로보트.06 가스
AND       P10609	// R06 Arc_On -> PLC
LOAD      P1060A	// R06 로보트 원위치
AND       P00015	// ARC 로보트.06 가스
AND NOT   P10609	// R06 Arc_On -> PLC
OR LOAD
AND LOAD
AND       P10606	// R06 PLAY Mode
AND NOT   D015013.6	// R06 GAS Check By_Pass On
TON       T2210 D000030	// R06 Gas On 검출이상 / 라인1 가스체크 설정시간
MPOP
LOAD      T2210	// R06 Gas On 검출이상
LOAD      M03910	// R06 Gas On 검출이상
AND NOT   M00004	// OP1 이상해제
AND NOT   M0000C	// OP2 이상해제
OR LOAD
AND LOAD
OUT       M03910	// R06 Gas On 검출이상
; L32
END

PROGRAM Data키핑 (task: 스캔 프로그램)

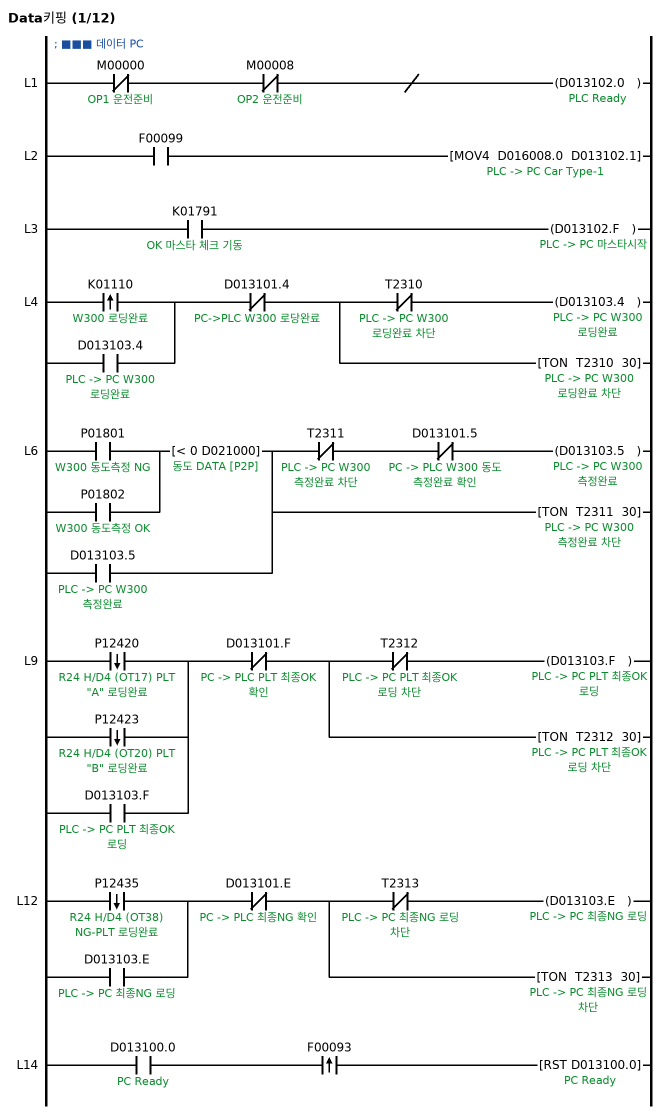
// ■■■ 데이터 PC
; L1
LOAD NOT  M00000	// OP1 운전준비
AND NOT   M00008	// OP2 운전준비
NOT
OUT       D013102.0	// PLC Ready
; L2
LOAD      F00099
MOV4      D016008.0 D013102.1	// PLC -> PC Car Type-1
; L3
LOAD      K01791	// OK 마스타 체크 기동
OUT       D013102.F	// PLC -> PC 마스타시작
; L4
LOADP     K01110	// W300 로딩완료
OR        D013103.4	// PLC -> PC W300 로딩완료
AND NOT   D013101.4	// PC->PLC W300 로당완료
MPUSH
AND NOT   T2310	// PLC -> PC W300 로딩완료 차단
OUT       D013103.4	// PLC -> PC W300 로딩완료
MPOP
TON       T2310 30	// PLC -> PC W300 로딩완료 차단
; L6
LOAD      P01801	// W300 동도측정 NG
OR        P01802	// W300 동도측정 OK
AND<      0 D021000	// 동도 DATA [P2P]
OR        D013103.5	// PLC -> PC W300 측정완료
MPUSH
AND NOT   T2311	// PLC -> PC W300 측정완료 차단
AND NOT   D013101.5	// PC -> PLC W300 동도 측정완료 확인
OUT       D013103.5	// PLC -> PC W300 측정완료
MPOP
TON       T2311 30	// PLC -> PC W300 측정완료 차단
; L9
LOADN     P12420	// R24 H/D4 (OT17) PLT "A" 로딩완료
ORN       P12423	// R24 H/D4 (OT20) PLT "B" 로딩완료
OR        D013103.F	// PLC -> PC PLT 최종OK 로딩
AND NOT   D013101.F	// PC -> PLC PLT 최종OK 확인
MPUSH
AND NOT   T2312	// PLC -> PC PLT 최종OK 로딩 차단
OUT       D013103.F	// PLC -> PC PLT 최종OK 로딩
MPOP
TON       T2312 30	// PLC -> PC PLT 최종OK 로딩 차단
; L12
LOADN     P12435	// R24 H/D4 (OT38) NG-PLT 로딩완료
OR        D013103.E	// PLC -> PC 최종NG 로딩
AND NOT   D013101.E	// PC -> PLC 최종NG 확인
MPUSH
AND NOT   T2313	// PLC -> PC 최종NG 로딩 차단
OUT       D013103.E	// PLC -> PC 최종NG 로딩
MPOP
TON       T2313 30	// PLC -> PC 최종NG 로딩 차단
; L14
LOAD      D013100.0	// PC Ready
ANDP      F00093
RST       D013100.0	// PC Ready

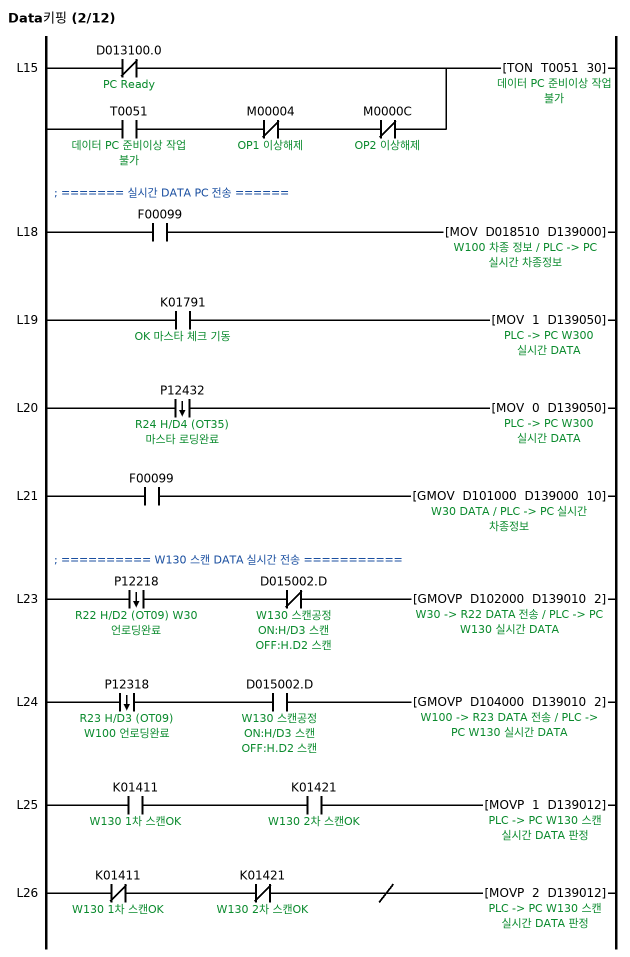
; L15
LOAD NOT  D013100.0	// PC Ready
LOAD      T0051	// 데이터 PC 준비이상 작업 불가
AND NOT   M00004	// OP1 이상해제
AND NOT   M0000C	// OP2 이상해제
OR LOAD
TON       T0051 30	// 데이터 PC 준비이상 작업 불가
// ======= 실시간 DATA PC 전송 ======
; L18
LOAD      F00099
MOV       D018510 D139000	// W100 차종 정보 / PLC -> PC 실시간 차종정보
; L19
LOAD      K01791	// OK 마스타 체크 기동
MOV       1 D139050	// PLC -> PC W300 실시간 DATA
; L20
LOADN     P12432	// R24 H/D4 (OT35) 마스타 로딩완료
MOV       0 D139050	// PLC -> PC W300 실시간 DATA
; L21
LOAD      F00099
GMOV      D101000 D139000 10	// W30 DATA / PLC -> PC 실시간 차종정보
// ========== W130 스캔 DATA 실시간 전송 ===========
; L23
LOADN     P12218	// R22 H/D2 (OT09) W30 언로딩완료
AND NOT   D015002.D	// W130 스캔공정 ON:H/D3 스캔 OFF:H.D2 스캔
GMOVP     D102000 D139010 2	// W30 -> R22 DATA 전송 / PLC -> PC W130 실시간 DATA
; L24
LOADN     P12318	// R23 H/D3 (OT09) W100 언로딩완료
AND       D015002.D	// W130 스캔공정 ON:H/D3 스캔 OFF:H.D2 스캔
GMOVP     D104000 D139010 2	// W100 -> R23 DATA 전송 / PLC -> PC W130 실시간 DATA
; L25
LOAD      K01411	// W130 1차 스캔OK
AND       K01421	// W130 2차 스캔OK
MOVP      1 D139012	// PLC -> PC W130 스캔 실시간 DATA 판정
; L26
LOAD NOT  K01411	// W130 1차 스캔OK
AND NOT   K01421	// W130 2차 스캔OK
NOT
MOVP      2 D139012	// PLC -> PC W130 스캔 실시간 DATA 판정

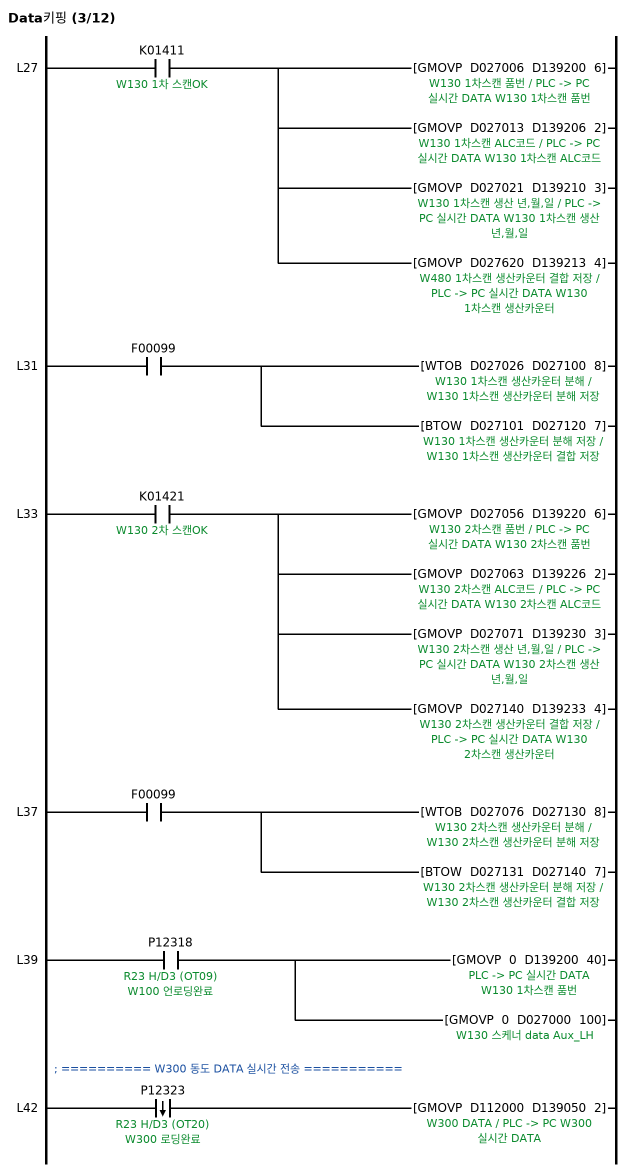
; L27
LOAD      K01411	// W130 1차 스캔OK
GMOVP     D027006 D139200 6	// W130 1차스캔 품번 / PLC -> PC 실시간 DATA W130 1차스캔 품번
GMOVP     D027013 D139206 2	// W130 1차스캔 ALC코드 / PLC -> PC 실시간 DATA W130 1차스캔 ALC코드
GMOVP     D027021 D139210 3	// W130 1차스캔 생산 년,월,일 / PLC -> PC 실시간 DATA W130 1차스캔 생산 년,월,일
GMOVP     D027620 D139213 4	// W480 1차스캔 생산카운터 결합 저장 / PLC -> PC 실시간 DATA W130 1차스캔 생산카운터
; L31
LOAD      F00099
WTOB      D027026 D027100 8	// W130 1차스캔 생산카운터 분해 / W130 1차스캔 생산카운터 분해 저장
BTOW      D027101 D027120 7	// W130 1차스캔 생산카운터 분해 저장 / W130 1차스캔 생산카운터 결합 저장
; L33
LOAD      K01421	// W130 2차 스캔OK
GMOVP     D027056 D139220 6	// W130 2차스캔 품번 / PLC -> PC 실시간 DATA W130 2차스캔 품번
GMOVP     D027063 D139226 2	// W130 2차스캔 ALC코드 / PLC -> PC 실시간 DATA W130 2차스캔 ALC코드
GMOVP     D027071 D139230 3	// W130 2차스캔 생산 년,월,일 / PLC -> PC 실시간 DATA W130 2차스캔 생산 년,월,일
GMOVP     D027140 D139233 4	// W130 2차스캔 생산카운터 결합 저장 / PLC -> PC 실시간 DATA W130 2차스캔 생산카운터
; L37
LOAD      F00099
WTOB      D027076 D027130 8	// W130 2차스캔 생산카운터 분해 / W130 2차스캔 생산카운터 분해 저장
BTOW      D027131 D027140 7	// W130 2차스캔 생산카운터 분해 저장 / W130 2차스캔 생산카운터 결합 저장
; L39
LOAD      P12318	// R23 H/D3 (OT09) W100 언로딩완료
GMOVP     0 D139200 40	// PLC -> PC 실시간 DATA W130 1차스캔 품번
GMOVP     0 D027000 100	// W130 스케너 data Aux_LH
// ========== W300 동도 DATA 실시간 전송 ===========
; L42
LOADN     P12323	// R23 H/D3 (OT20) W300 로딩완료
GMOVP     D112000 D139050 2	// W300 DATA / PLC -> PC W300 실시간 DATA

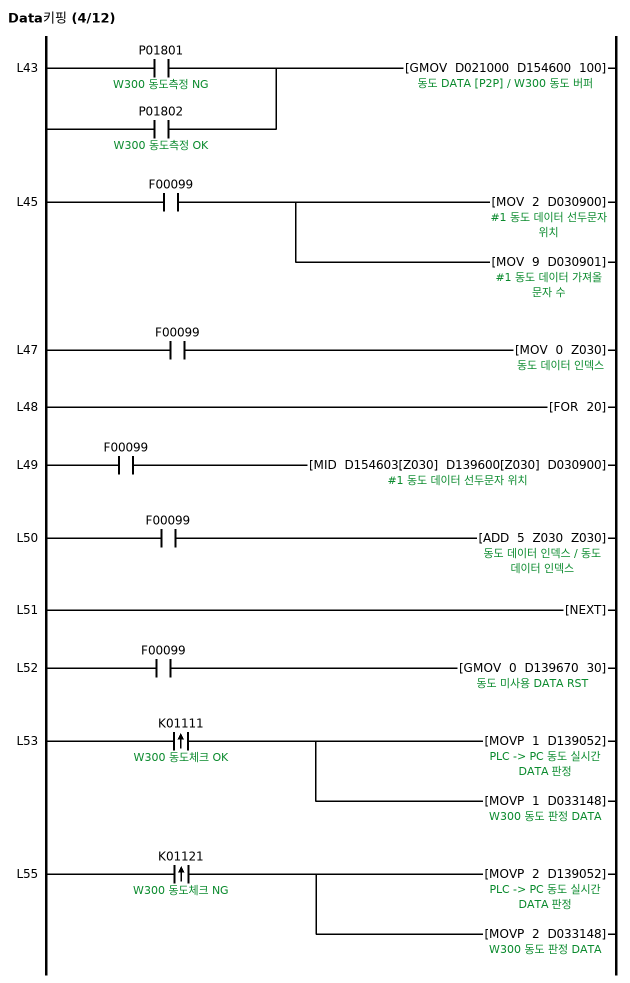
; L43
LOAD      P01801	// W300 동도측정 NG
OR        P01802	// W300 동도측정 OK
GMOV      D021000 D154600 100	// 동도 DATA [P2P] / W300 동도 버퍼
; L45
LOAD      F00099
MOV       2 D030900	// #1 동도 데이터 선두문자 위치
MOV       9 D030901	// #1 동도 데이터 가져올 문자 수
; L47
LOAD      F00099
MOV       0 Z030	// 동도 데이터 인덱스
; L48
FOR       20
; L49
LOAD      F00099
MID       D154603[Z030] D139600[Z030] D030900	// #1 동도 데이터 선두문자 위치
; L50
LOAD      F00099
ADD       5 Z030 Z030	// 동도 데이터 인덱스 / 동도 데이터 인덱스
; L51
NEXT
; L52
LOAD      F00099
GMOV      0 D139670 30	// 동도 미사용 DATA RST
; L53
LOADP     K01111	// W300 동도체크 OK
MOVP      1 D139052	// PLC -> PC 동도 실시간 DATA 판정
MOVP      1 D033148	// W300 동도 판정 DATA
; L55
LOADP     K01121	// W300 동도체크 NG
MOVP      2 D139052	// PLC -> PC 동도 실시간 DATA 판정
MOVP      2 D033148	// W300 동도 판정 DATA

